FUNCTION_BLOCK deneme
VAR_INPUT//girilecek değerler
	bEnable			: BOOL;
	fPosition1		: LREAL;
	fPosition2		: LREAL;
	fVelocity		: LREAL;
	tDelay 			: TIME;
END_VAR
VAR_OUTPUT
	bError			: BOOL;
	sStatus 		: STRING;
END_VAR
VAR//kullanıcının görmesine gerek yok!
	fbPower 		: MC_Power;
	fbPower2		: MC_Power;
	fbMove 			: MC_MoveAbsolute;
	fbMove2			: MC_MoveAbsolute;
	nState 			: INT;
	fbTimer 		: TON;
END_VAR

VAR_IN_OUT 
	Axis 		:AXIS_REF;
	Axis2		:AXIS_REF;
END_VAR

fbPower2(
	Axis:= Axis2, 
	Enable:= TRUE, 
	Enable_Positive:= TRUE, 
	Enable_Negative:= TRUE, 
	Override:=  100);
fbMove2(
	Axis:= Axis2, 
	Velocity:=fVelocity , 
);
fbPower(
	Axis:= Axis, 
	Enable:= TRUE , 
	Enable_Positive:= TRUE, 
	Enable_Negative:= TRUE, 
	Override:=100);
	
	fbMove(
	Axis:= Axis, 
	Velocity:= fVelocity);
	
	Axis.ReadStatus();
	Axis2.ReadStatus();
	
	fbTimer(PT:= tDelay);
	CASE nState OF
	0://eksen enable state
			bError:=FALSE;
			sStatus :='Beklemede';
			IF bEnable AND Axis.Status.Operational AND Axis2.Status.Operational THEN
				nState :=10;
				ELSIF NOT  Axis.Status.Operational OR Axis2.Status.Operational THEN
					nState :=900;
					sStatus :='Enable değil';
			END_IF
			
	10://Execute state'i.
		fbMove.Position:=fPosition1;
		fbMove2.Position:=fPosition2;
		fbMove.Execute:=TRUE;
		IF Axis.Status.Moving AND Axis2.Status.Moving THEN
			sStatus 	:='Eksenler ilk noktaya Hareket ediyor.';
			nState:=20;
			ELSIF Axis.Status.Error OR fbMove.Error OR Axis2.Status.Error OR fbMove2.Error  THEN
				sStatus :='1. noktaya giderken hataya geçti';
				nState :=900;
		END_IF
			
	20://hareket kontrol state'i.
		IF fbMove.Done AND fbMove2.Done THEN
			sStatus 		:='1. Noktaya vardı';
			nState 			:=30;
			fbMove.Execute:=FALSE;//2. hareket için false'a çektik.
			fbMove2.Execute:=FALSE;
			
		END_IF
		
	30: //timer state
		fbTimer.IN:= TRUE;
		sStatus:='1. Noktada bekliyor.';
		IF(fbTimer.Q) THEN
			fbTimer.IN:=FALSE;
			nState :=40;
			
		END_IF
	40://2. noktaya hareket.
		fbMove2.Position:=fPosition2;
		fbMove.Position:=fPosition1;
		fbMove.Execute:=TRUE;
		fbMove2.Execute:=TRUE;
		IF Axis.Status.Moving AND Axis2.Status.Moving THEN
			sStatus :='2. noktaya hareket ediyor';
			nState := 50;
		ELSIF  Axis.Status.Error OR fbMove.Error OR Axis2.Status.Error OR fbMove2.Error THEN
			sStatus :='2. noktaya geçerken hataya geçti';
			nState :=900;
		END_IF
	50:
		IF fbMove.Done AND fbMove2.Done THEN
			sStatus :='2. noktaya vardı.';
			nstate :=60;
			fbMove.Execute:=FALSE;
			
		END_IF
	60:
		fbTimer.IN:=TRUE;
		sStatus :='2. noktada bekliyor';
		IF fbTimer.Q THEN
			fbTimer.IN:=FALSE;			
			nState :=0;
		END_IF
	900:
		bError := TRUE;
		IF NOT bEnable THEN
			fbTimer(IN:=FALSE);
			nState:=0;
		END_IF
		
	END_CASE

END_FUNCTION_BLOCK

(* stored: Version 1.1.0.1, ProductVersion 3.1.4024.12
   POU deneme: Id {c9c82607-25ec-4aa3-b1f6-505ff7513975}, SpecialFunc None *)
